FUNCTION_BLOCK FB_CasingVibratoryBowl1
VAR_INPUT
END_VAR
VAR_OUTPUT
END_VAR
VAR
    iState : INT := 0;
    iState2 : INT := 0;
	FeedbackTimer : TON;
    DelayTimer : TON;
	DelayTimer2 : TON;
END_VAR

IF GVL_HMI.i_nCmd_ClearCount = 2 THEN
	GVL_HMI.nCasingCount := 0;
END_IF

CASE iState OF
    0: (* Idle/Off *)
		iState := 10;
	
	10:
        IF GVL_HMI.bSafeties AND GVL_IO.DI_ECS THEN
            iState := iState + 10;
        END_IF

    20: (* Wait for Product in Position *)
		DelayAndAdvance( GVL_InitialSetting.BOWL_RunningDelayTime, iState+1 );
	21:
	    IF GVL_IO.DI_PE1 THEN
            iState := (iState + 10) / 10 * 10;
        END_IF

    30: (* Energize Track Index Solenoid *)
        GVL_IO.DO_PCYL3_E := TRUE;
		DelayAndAdvance( GVL_HMI.i_nPCylinder3ExtendedRunningTime, iState+1 );
	31:
		GVL_IO.DO_PCYL3_E := FALSE;
		iState2 := 0;
        iState := (iState + 10) / 10 * 10;
		
	40:
		DelayAndAdvance( GVL_InitialSetting.PE2_CheckingDelayTime, iState+1 );
	41: (* Check Invert PE and Decide Path *)
		IF GVL_IO.DI_PE2 THEN
			iState := iState + 10;
			DelayTimer.IN := FALSE;
		ELSE
			DelayAndAdvance( GVL_InitialSetting.PE2_MaintainTime, iState+20 );
		END_IF
	
	50:
		GVL_IO.DO_PCYL5_E := TRUE;
		DelayAndAdvance( GVL_HMI.i_nPCylinder5ExtendedRunningTime, iState+1);
	51:
		GVL_IO.DO_PCYL5_E := FALSE;
		GVL_HMI.nCasingCount := GVL_HMI.nCasingCount + 1;
		iState := 20;
		
	60:
		GVL_IO.DO_PCYL4_E := TRUE;
		DelayAndAdvance( GVL_HMI.i_nPCylinder4ExtendedRunningTime, iState+1);
	61:
		GVL_IO.DO_PCYL4_E := FALSE;
		GVL_HMI.nCasingCount := GVL_HMI.nCasingCount + 1;
		iState := (iState + 10) / 10 * 10;
		
	70: (* Check High-Level Sensor *)
		IF GVL_IO.DI_PE4 THEN
			DelayAndAdvance( GVL_HMI.i_nPE4MaintainTime, iState+10 );
		ELSE
			iState := 20;
			DelayTimer.IN := FALSE;
		END_IF
	
	80:
		(* Pause and Wait *)
END_CASE

IF iState >= 20 THEN
	CASE iState2 OF
		0:
			GVL_IO.DO_VB1 := TRUE; 
			IF NOT DelayTimer2.IN THEN
				DelayTimer2(IN := TRUE, PT := INT_TO_TIME(GVL_InitialSetting.VB1_MaintainTime));
			ELSE
				IF DelayTimer2.Q THEN 
					iState2 := iState2 + 10;
				END_IF
			END_IF
		10:
			IF GVL_IO.DI_PE1 THEN
				iState2 := iState2 + 10;
			END_IF
		20:
			(* Stop and Wait *)
	END_CASE
ELSE
	iState2 := 0;
END_IF

METHOD DelayAndAdvance : BOOL
VAR_INPUT
	i_nDelayTime: INT;	// ms
	i_nNextState: INT;
END_VAR

VAR
END_VAR
IF NOT DelayTimer.IN THEN
    DelayTimer(IN := TRUE, PT := INT_TO_TIME(i_nDelayTime));
ELSE
    IF DelayTimer.Q THEN 
        iState := i_nNextState; 
    END_IF
END_IF
END_METHOD

END_FUNCTION_BLOCK

(* stored: Version 1.1.0.1, ProductVersion 3.1.4024.11
   POU FB_CasingVibratoryBowl1: Id {964fa243-99d7-4cd8-a60f-98887c839cc0}, SpecialFunc None
   Method DelayAndAdvance: Id {41bcb24e-3142-49ab-9a22-b6668bf4ec63} *)
